VAR_GLOBAL
	
	XTags			: ST_XTags;		

	stVisControl	: ST_VisControl;
	

END_VAR

(* stored: Version 1.1.0.1, ProductVersion 3.1.4024.3
   GVL GlobalVariables: Id {13561444-0093-44b8-8531-b64033cc874c} *)
